// Mitsubishi GX Works2 project: PLC_Group7 Finishhh   PLC: FX3G

// global labels: Global1
VAR_GLOBAL
  Start_Day AT X007 : BOOL;
  Emergency_Switch AT X005 : BOOL;
  LackMaterials AT M1 : BOOL;
  Work_Day AT Y007 : BOOL;
  Y7coil AT Y007 : BOOL;
  EndDayReset AT M2 : BOOL;
  Chocolate_Input AT D1100 : REAL;
  Chocolate_Stock AT D1101 : REAL;
  Nuts_Input AT D1102 : REAL;
  Nuts_Stock AT D1103 : REAL;
  Fistock_Input AT D1104 : REAL;
  Fistock_Stock AT D1105 : REAL;
  Kadaif_Input AT D1106 : REAL;
  Kadaif_Stock AT D1107 : REAL;
  Chocolate_Package AT D1108 : REAL;
  Start_Melting AT X001 : BOOL;
  Min_Chocolate AT E400 : REAL;
  Check_Chocolate AT M3 : BOOL;
  Chocolate_Melting_Tank AT D1110 : REAL;
  Temp_Sensor AT X002 : BOOL;
  End_Melting AT Y001 : BOOL;
  Flag_End_Melting AT M4 : BOOL;
  Location_Sensor AT X003 : BOOL;
  Flag_End_Location AT M5 : BOOL;
  MoldCastingTimer AT TC1 : BOOL;
  MoldCasting AT K40 : INT;
  FinishCasting AT TS1 : BOOL;
  InCastingProcess AT Y002 : BOOL;
  Empty_Mold_Tank AT D1114 : REAL;
  Flag_End_Casting AT M6 : BOOL;
  Chocolate_Type AT X004 : BOOL;
  Make_Nuts_Chocolate AT M7 : BOOL;
  Nuts_N AT E100 : REAL;
  Fistock_N AT E100 : REAL;
  Kadaif_N AT E0 : REAL;
  Out_Of_Stock_Nuts AT M9 : BOOL;
  Choose_Type AT X004 : BOOL;
  Dubai_Chocolate AT M8 : BOOL;
  Nuts_D AT E20 : REAL;
  Fistock_D AT E120 : REAL;
  Kadaif_D AT E60 : REAL;
  Out_Of_Stock_Dubai AT M10 : BOOL;
  Start_Making AT X004 : BOOL;
END_VAR
VAR_GLOBAL CONSTANT
  Convert : REAL := 400;
END_VAR
VAR_GLOBAL
  Chocolate_Ch AT D7000 : REAL;
  Chocolate_Choice AT D7000 : REAL;
  Choose_Nuts AT E5 : REAL;
  Make_Dubai_Chocolate AT M8 : BOOL;
  Min_Amount_Nuts_D AT E10 : REAL;
  Amount_Cream_Nuts AT E50 : REAL;
  Cream_Tank_Nuts AT D1116 : REAL;
  Cream_Tank_Dubi AT D1118 : REAL;
  Amount_Cream_Dubai AT E50 : REAL;
  Cream_Tank_Dubai AT D1118 : REAL;
  Start_Cream AT M11 : BOOL;
  Start_Flash AT TC2 : BOOL;
  Finish_Flesh AT TS2 : BOOL;
  Start_Flashing AT M12 : BOOL;
  Timer_Flash AT K50 : INT;
  Flech3 AT TC3 : BOOL;
  Flesh_CreaFill3 AT Y003 : BOOL;
  Finish_Flesh3 AT TS3 : BOOL;
  Flesh4 AT TC4 : BOOL;
  Finish_Flesh4 AT TS4 : BOOL;
  Flesh_CreamFill4 AT Y004 : BOOL;
  Flesh_CreamFill3 AT Y003 : BOOL;
  Time_Flesh34 AT K5 : INT;
  Melting AT Y001 : BOOL;
  Freeze_Chocolate AT X006 : BOOL;
  Time_Freeze AT TC5 : BOOL;
  Three_Sec_Freeze AT K30 : INT;
  Freeze_Light AT Y006 : BOOL;
  Finish_Freeze AT TS5 : BOOL;
  Start_Packing AT X006 : BOOL;
  Chocolate_Counter AT CC1 : BOOL;
  Chocolate_Package_Counter AT CC1 : BOOL;
END_VAR
VAR_GLOBAL CONSTANT
  Four_Package_Chocolate : INT := K4;
END_VAR
VAR_GLOBAL
  Packing_One AT X000 : BOOL;
  Pack_Light AT Y005 : BOOL;
  CS_Packing AT CS1 : BOOL;
  Counter_1 AT K1 : INT;
  Package_Number AT D4000 : REAL;
  Package_Number_Output : INT;
END_VAR
VAR_GLOBAL CONSTANT
  PI : INT := 40;
END_VAR
VAR_GLOBAL
  Analog_Output AT D8282 : INT;
  Insert_Stock AT M14 : BOOL;
  Analog_Input AT D8280 : INT;
  Analog_Input1 AT D8280 : INT;
  Choose_Nuts1 AT E5 : REAL;
  Amount_Cream_Dubai1 AT E200 : REAL;
  Amount_Cream_Nuts1 AT E200 : REAL;
  Flash_Help AT M15 : BOOL;
END_VAR
VAR_GLOBAL CONSTANT
  PI1 : INT := 40;
END_VAR
VAR_GLOBAL
  Out_Of_Stock AT M9 : BOOL;
END_VAR
VAR_GLOBAL CONSTANT
  Zero : REAL;
END_VAR
VAR_GLOBAL
  Reset_Data AT X010 : BOOL;
END_VAR

// task Task_01 (event TRUE, interval 0, priority 31): POU_01

PROGRAM POU_01
(* structured ladder/FBD written out as ST: instructions are called as NAME(EN, inputs, outputs); _pN, _eN, _tN stand for wires *)
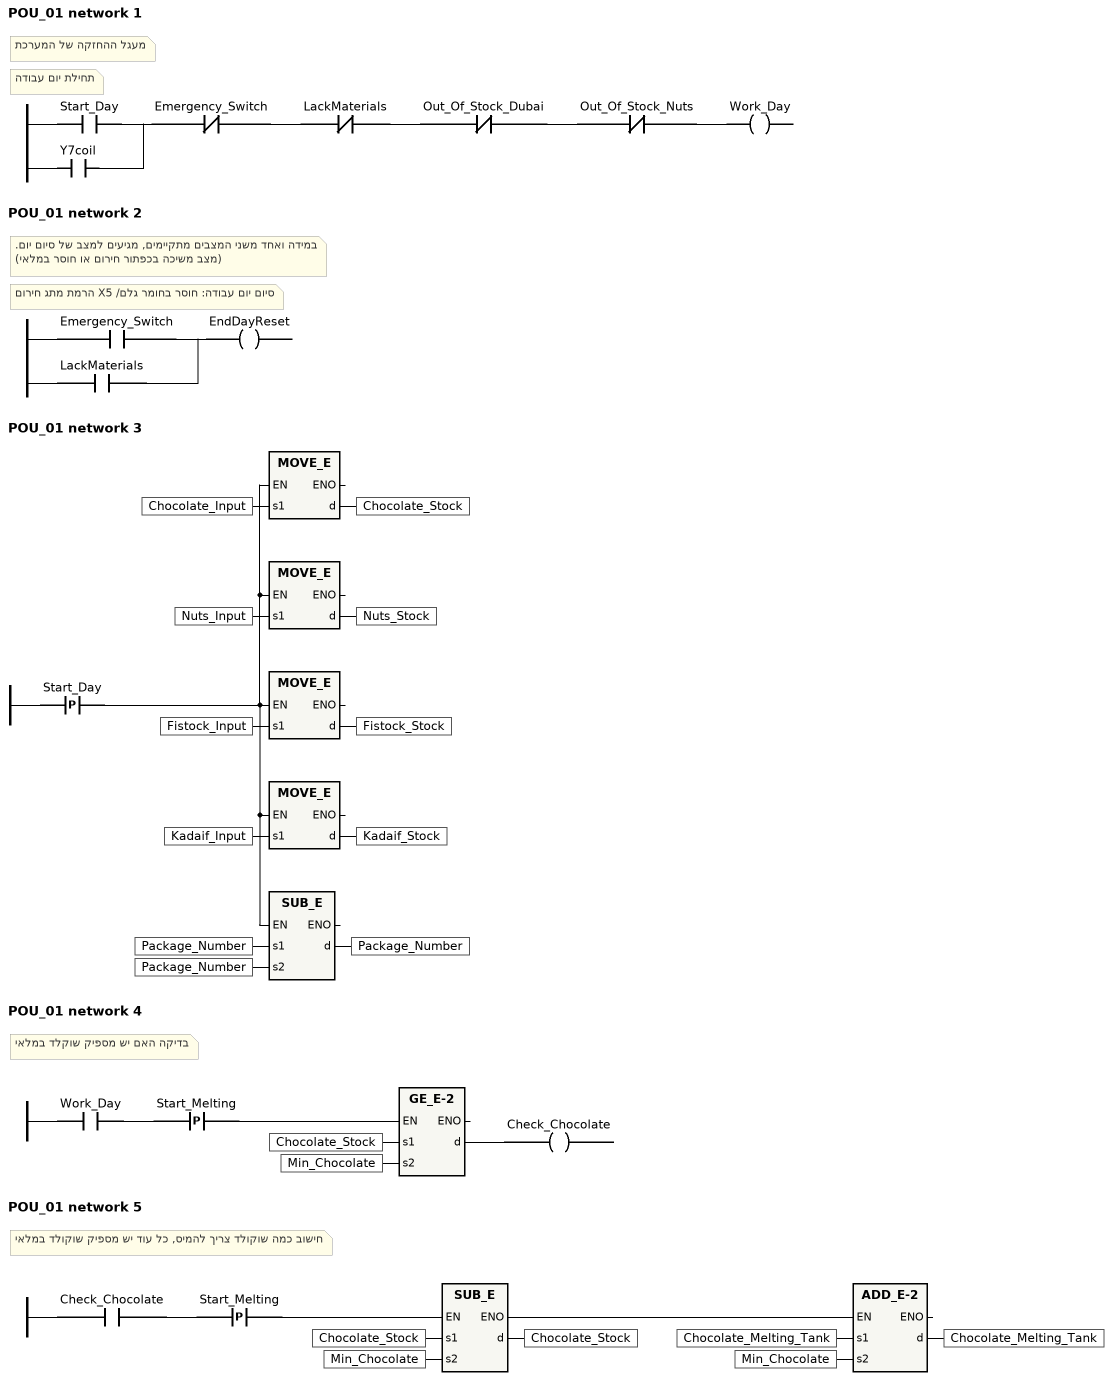
(* network 1 מעגל ההחזקה של המערכ *)
(* מעגל ההחזקה של המערכת *)
(* תחילת יום עבודה *)
Work_Day := ((((Start_Day OR Y7coil) AND NOT Emergency_Switch) AND NOT LackMaterials) AND NOT Out_Of_Stock_Dubai) AND NOT Out_Of_Stock_Nuts;
(* network 2 *)
(* במידה ואחד משני המצבים מתקיימים, מגיעים למצב של סיום יום. (מצב משיכה בכפתור חירום או חוסר במלאי) *)
(* סיום יום עבודה: חוסר בחומר גלם/ X5 הרמת מתג חירום *)
EndDayReset := Emergency_Switch OR LackMaterials;
(* network 3 *)
_p1 := LDP(TRUE, Start_Day);
MOVE_E(_p1, Chocolate_Input, Chocolate_Stock);
MOVE_E(_p1, Nuts_Input, Nuts_Stock);
MOVE_E(_p1, Fistock_Input, Fistock_Stock);
MOVE_E(_p1, Kadaif_Input, Kadaif_Stock);
SUB_E(_p1, Package_Number, Package_Number, Package_Number);
(* network 4 *)
(* בדיקה האם יש מספיק שוקלד במלאי *)
GE_E(Work_Day AND LDP(TRUE, Start_Melting), Chocolate_Stock, Min_Chocolate, _t1);
Check_Chocolate := _t1;
(* network 5 *)
(* חישוב כמה שוקולד צריך להמיס, כל עוד יש מספיק שוקולד במלאי *)
_e1 := SUB_E(Check_Chocolate AND LDP(TRUE, Start_Melting), Chocolate_Stock, Min_Chocolate, Chocolate_Stock);
ADD_E(_e1, Chocolate_Melting_Tank, Min_Chocolate, Chocolate_Melting_Tank);
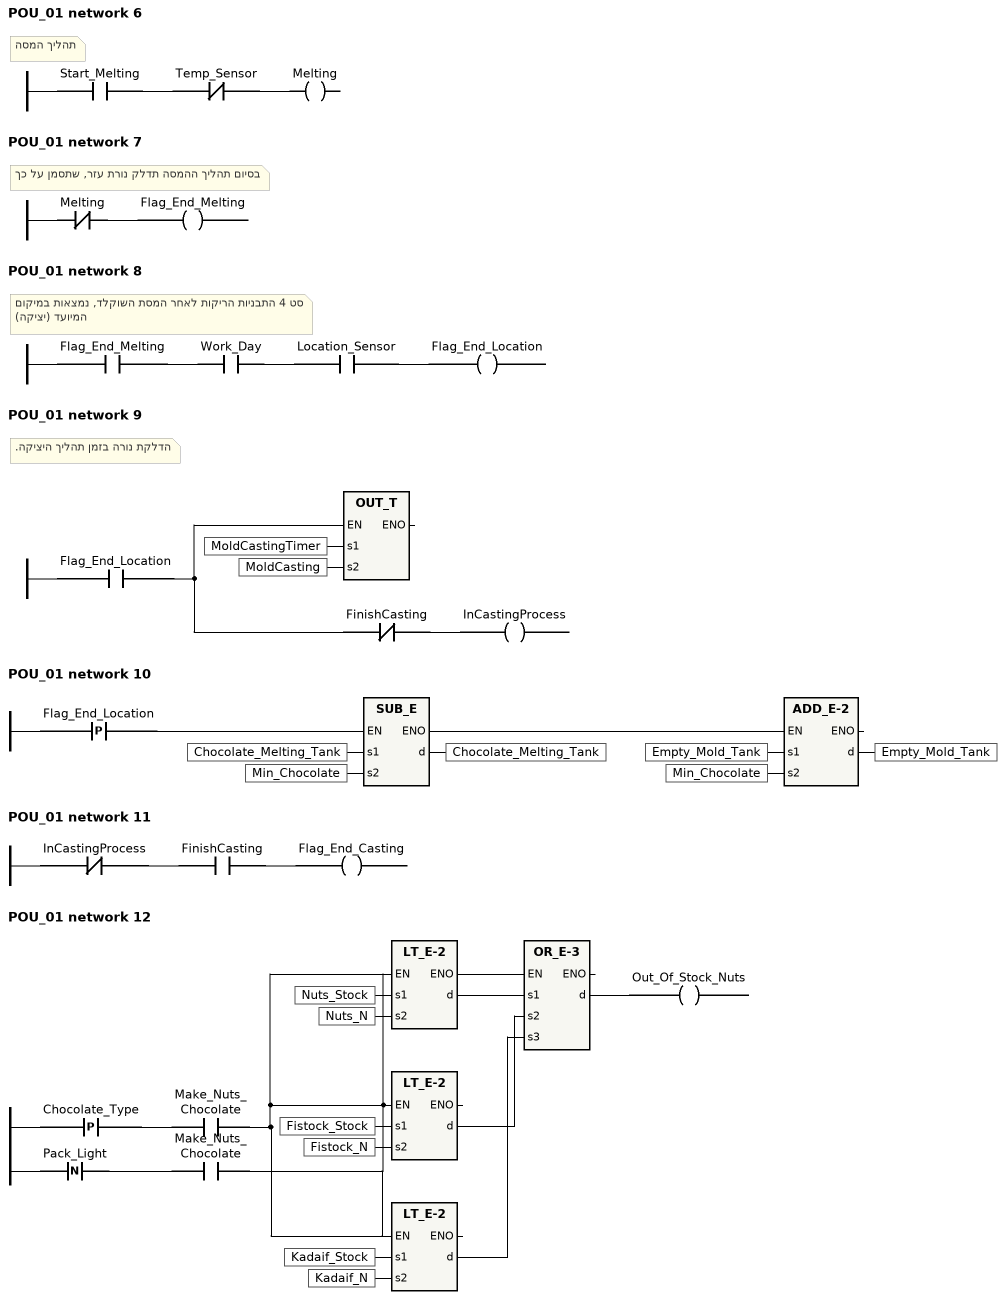
(* network 6 *)
(* תהליך המסה *)
Melting := Start_Melting AND NOT Temp_Sensor;
(* network 7 *)
(* בסיום תהליך ההמסה תדלק נורת עזר, שתסמן על כך *)
Flag_End_Melting := NOT Melting;
(* network 8 *)
(* סט 4 התבניות הריקות לאחר המסת השוקלד, נמצאות במיקום המיועד (יציקה) *)
Flag_End_Location := Flag_End_Melting AND Work_Day AND Location_Sensor;
(* network 9 *)
(* הדלקת נורה בזמן תהליך היציקה. *)
OUT_T(Flag_End_Location, MoldCastingTimer, MoldCasting);
InCastingProcess := Flag_End_Location AND NOT FinishCasting;
(* network 10 *)
_e1 := SUB_E(LDP(TRUE, Flag_End_Location), Chocolate_Melting_Tank, Min_Chocolate, Chocolate_Melting_Tank);
ADD_E(_e1, Empty_Mold_Tank, Min_Chocolate, Empty_Mold_Tank);
(* network 11 *)
Flag_End_Casting := NOT InCastingProcess AND FinishCasting;
(* network 12 *)
_p1 := (LDP(TRUE, Chocolate_Type) AND Make_Nuts_Chocolate) OR (LDF(TRUE, Pack_Light) AND Make_Nuts_Chocolate);
_e3 := LT_E(_p1, Nuts_Stock, Nuts_N, _t2);
LT_E(_p1, Fistock_Stock, Fistock_N, _t4);
LT_E(_p1, Kadaif_Stock, Kadaif_N, _t5);
OR_E(_e3, _t2, _t4, _t5, _t6);
Out_Of_Stock_Nuts := _t6;
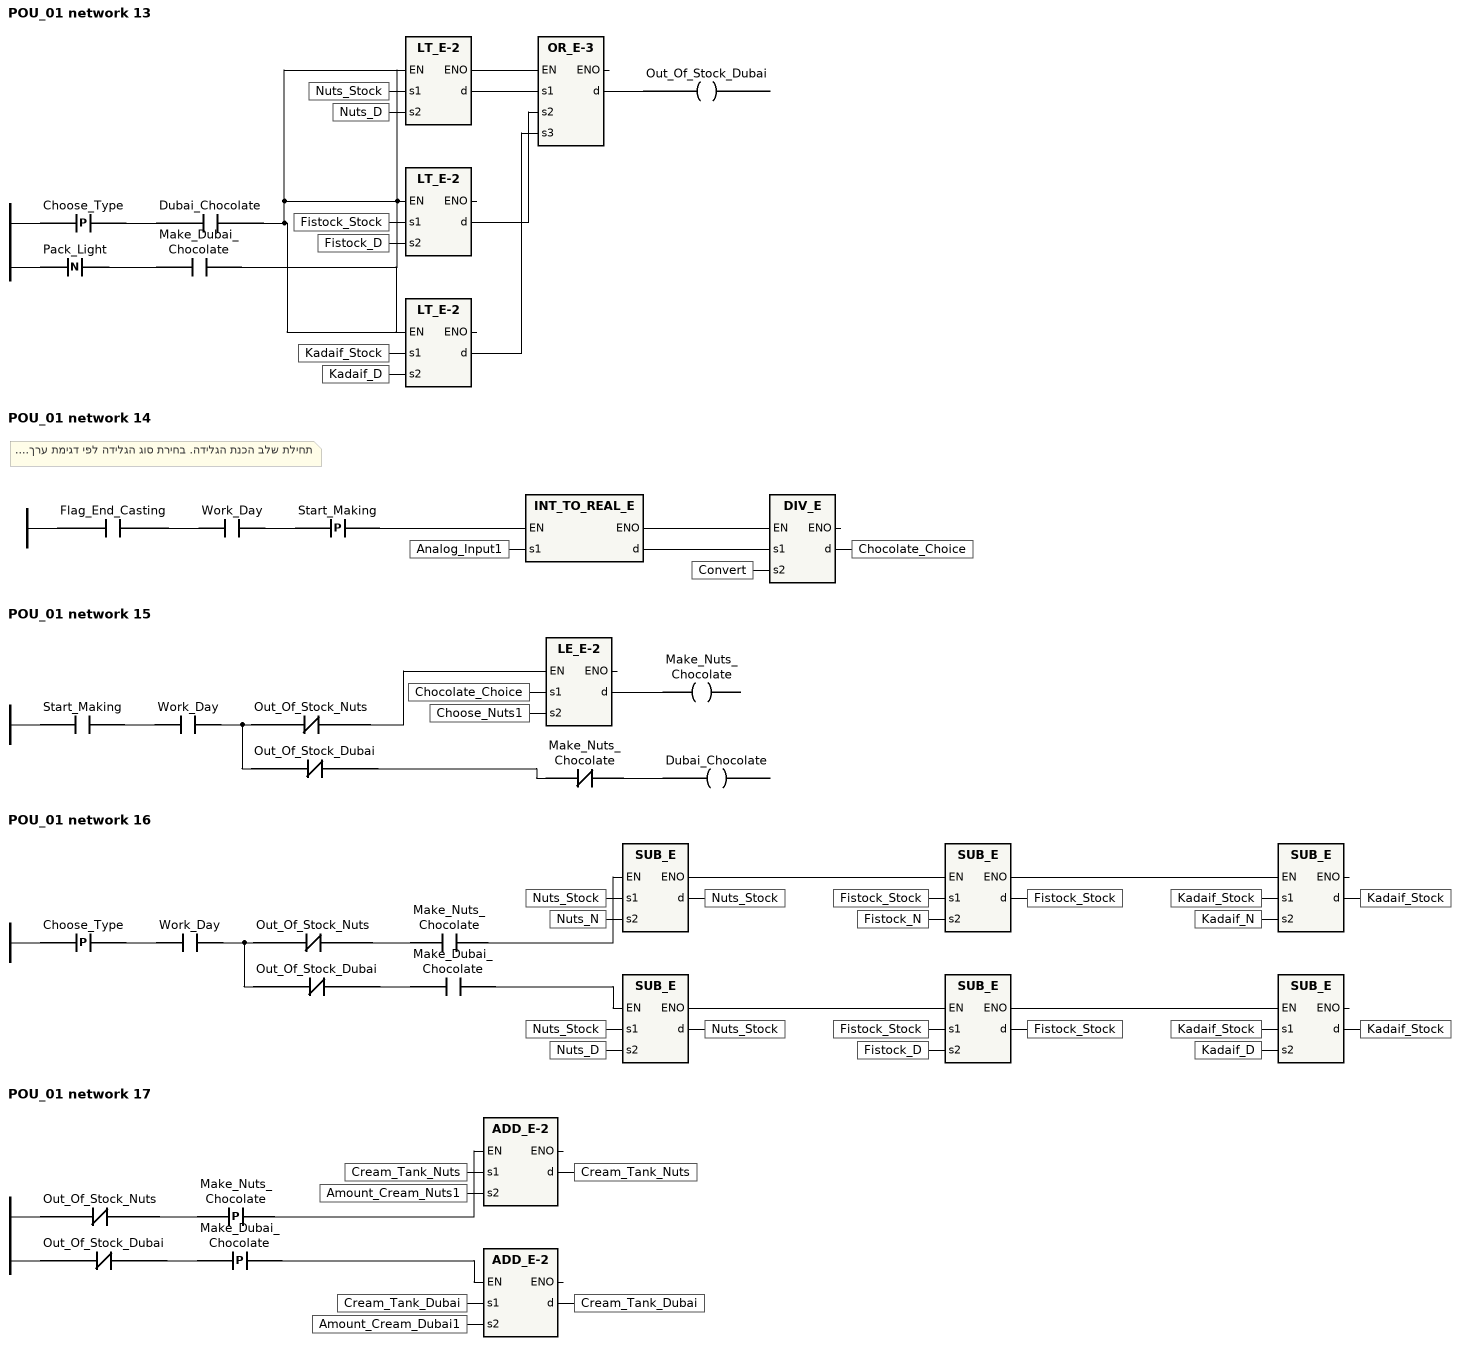
(* network 13 *)
_p1 := (LDP(TRUE, Choose_Type) AND Dubai_Chocolate) OR (LDF(TRUE, Pack_Light) AND Make_Dubai_Chocolate);
_e3 := LT_E(_p1, Nuts_Stock, Nuts_D, _t2);
LT_E(_p1, Fistock_Stock, Fistock_D, _t4);
LT_E(_p1, Kadaif_Stock, Kadaif_D, _t5);
OR_E(_e3, _t2, _t4, _t5, _t6);
Out_Of_Stock_Dubai := _t6;
(* network 14 *)
(* תחילת שלב הכנת הגלידה. בחירת סוג הגלידה לפי דגימת ערך.... *)
_e2 := INT_TO_REAL_E(Flag_End_Casting AND Work_Day AND LDP(TRUE, Start_Making), Analog_Input1, _t1);
DIV_E(_e2, _t1, Convert, Chocolate_Choice);
(* network 15 *)
_p1 := Start_Making AND Work_Day;
LE_E(_p1 AND NOT Out_Of_Stock_Nuts, Chocolate_Choice, Choose_Nuts1, _t2);
Make_Nuts_Chocolate := _t2;
Dubai_Chocolate := _p1 AND NOT Out_Of_Stock_Dubai AND NOT Make_Nuts_Chocolate;
(* network 16 *)
_p1 := LDP(TRUE, Choose_Type) AND Work_Day;
_e2 := SUB_E(_p1 AND NOT Out_Of_Stock_Nuts AND Make_Nuts_Chocolate, Nuts_Stock, Nuts_N, Nuts_Stock);
_e3 := SUB_E(_e2, Fistock_Stock, Fistock_N, Fistock_Stock);
SUB_E(_e3, Kadaif_Stock, Kadaif_N, Kadaif_Stock);
_e4 := SUB_E(_p1 AND NOT Out_Of_Stock_Dubai AND Make_Dubai_Chocolate, Nuts_Stock, Nuts_D, Nuts_Stock);
_e5 := SUB_E(_e4, Fistock_Stock, Fistock_D, Fistock_Stock);
SUB_E(_e5, Kadaif_Stock, Kadaif_D, Kadaif_Stock);
(* network 17 *)
ADD_E(NOT Out_Of_Stock_Nuts AND LDP(TRUE, Make_Nuts_Chocolate), Cream_Tank_Nuts, Amount_Cream_Nuts1, Cream_Tank_Nuts);
ADD_E(NOT Out_Of_Stock_Dubai AND LDP(TRUE, Make_Dubai_Chocolate), Cream_Tank_Dubai, Amount_Cream_Dubai1, Cream_Tank_Dubai);
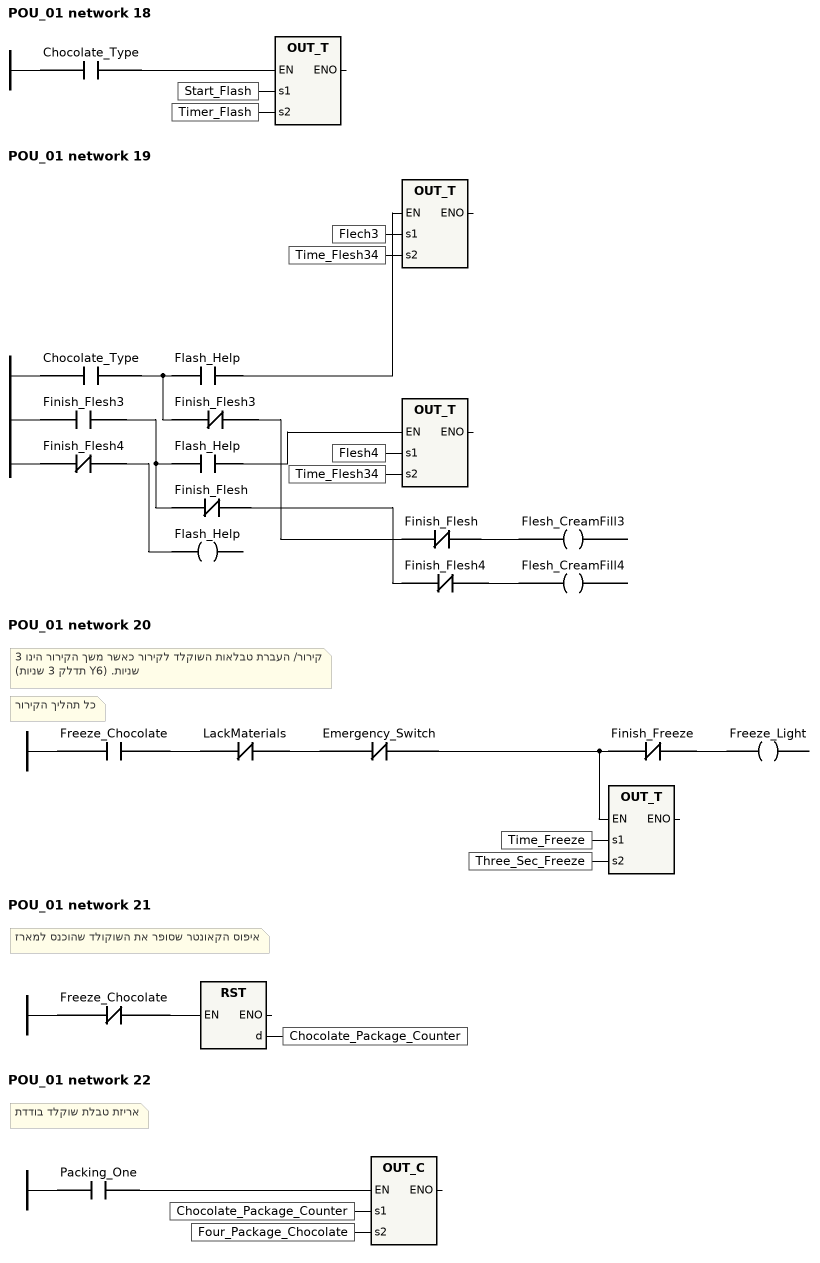
(* network 18 *)
OUT_T(Chocolate_Type, Start_Flash, Timer_Flash);
(* network 19 *)
OUT_T(Chocolate_Type AND Flash_Help, Flech3, Time_Flesh34);
Flesh_CreamFill3 := Chocolate_Type AND NOT Finish_Flesh3 AND NOT Finish_Flesh;
OUT_T(Finish_Flesh3 AND Flash_Help, Flesh4, Time_Flesh34);
Flesh_CreamFill4 := Finish_Flesh3 AND NOT Finish_Flesh AND NOT Finish_Flesh4;
Flash_Help := NOT Finish_Flesh4;
(* network 20 *)
(* קירור/ העברת טבלאות השוקלד לקירור כאשר משך הקירור הינו 3 שניות. (Y6 תדלק 3 שניות) *)
(* כל תהליך הקירור *)
_p1 := Freeze_Chocolate AND NOT LackMaterials AND NOT Emergency_Switch;
Freeze_Light := _p1 AND NOT Finish_Freeze;
OUT_T(_p1, Time_Freeze, Three_Sec_Freeze);
(* network 21 *)
(* איפוס הקאונטר שסופר את השוקולד שהוכנס למארז *)
RST(NOT Freeze_Chocolate, Chocolate_Package_Counter);
(* network 22 *)
(* אריזת טבלת שוקלד בודדת *)
OUT_C(Packing_One, Chocolate_Package_Counter, Four_Package_Chocolate);
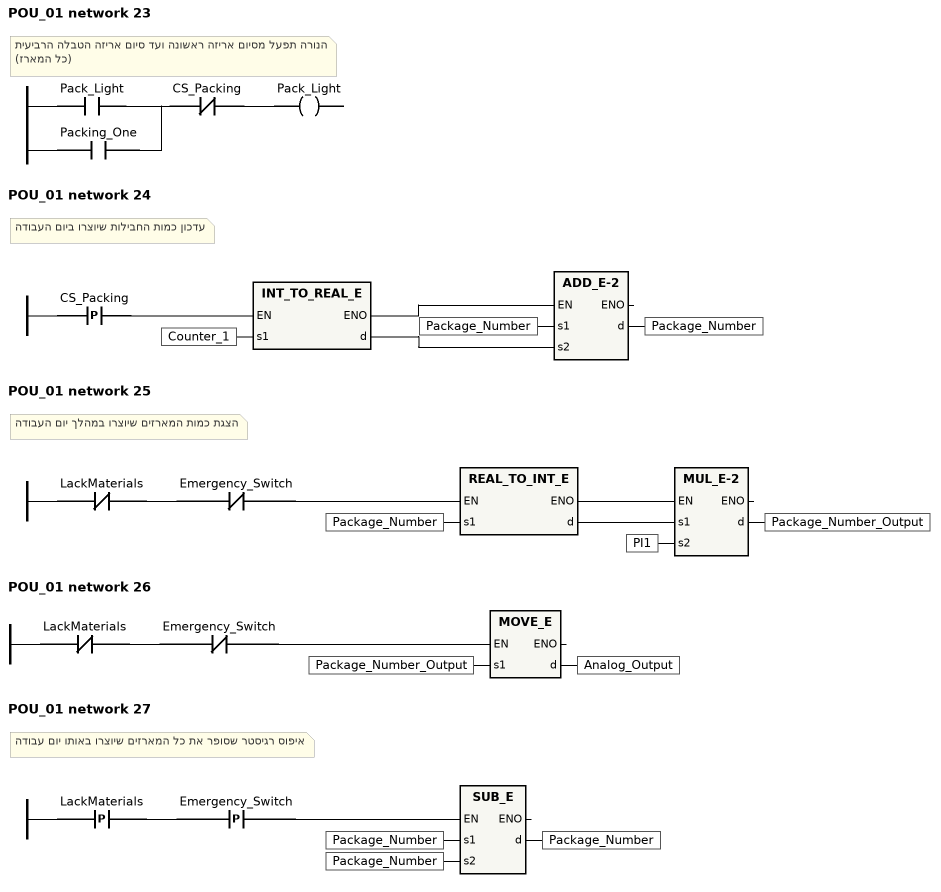
(* network 23 *)
(* הנורה תפעל מסיום אריזה ראשונה ועד סיום אריזה הטבלה הרביעית (כל המארז) *)
Pack_Light := (Pack_Light OR Packing_One) AND NOT CS_Packing;
(* network 24 *)
(* עדכון כמות החבילות שיוצרו ביום העבודה *)
_e2 := INT_TO_REAL_E(LDP(TRUE, CS_Packing), Counter_1, _t1);
ADD_E(_e2, Package_Number, _t1, Package_Number);
(* network 25 *)
(* הצגת כמות המארזים שיוצרו במהלך יום העבודה *)
_e2 := REAL_TO_INT_E(NOT LackMaterials AND NOT Emergency_Switch, Package_Number, _t1);
MUL_E(_e2, _t1, PI1, Package_Number_Output);
(* network 26 *)
MOVE_E(NOT LackMaterials AND NOT Emergency_Switch, Package_Number_Output, Analog_Output);
(* network 27 *)
(* איפוס רגיסטר שסופר את כל המארזים שיוצרו באותו יום עבודה *)
SUB_E(LDP(TRUE, LackMaterials) AND LDP(TRUE, Emergency_Switch), Package_Number, Package_Number, Package_Number);
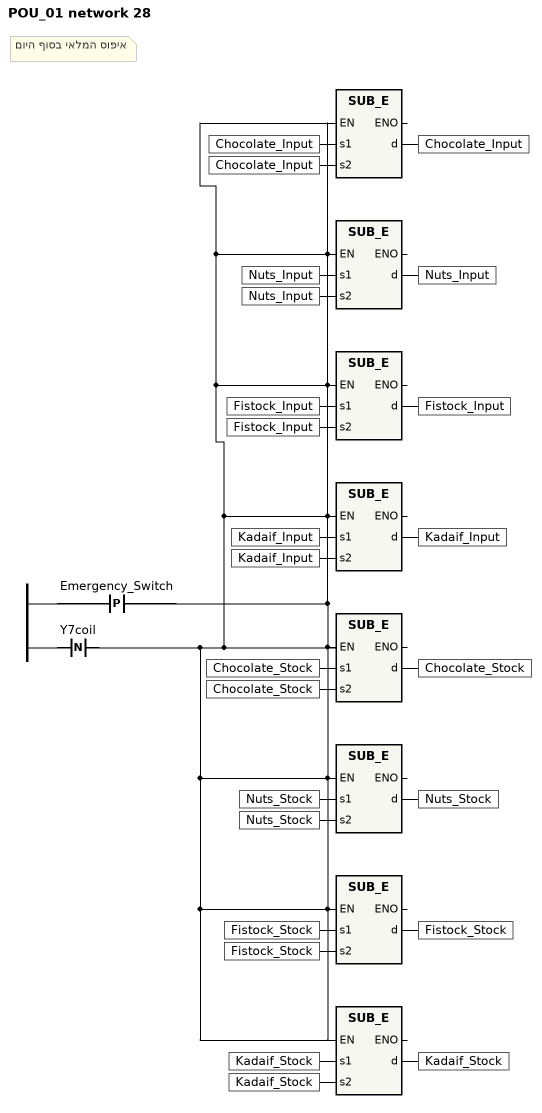
(* network 28 *)
(* איפוס המלאי בסוף היום *)
_p1 := LDP(TRUE, Emergency_Switch) OR LDF(TRUE, Y7coil);
SUB_E(_p1, Chocolate_Input, Chocolate_Input, Chocolate_Input);
SUB_E(_p1, Nuts_Input, Nuts_Input, Nuts_Input);
SUB_E(_p1, Fistock_Input, Fistock_Input, Fistock_Input);
SUB_E(_p1, Kadaif_Input, Kadaif_Input, Kadaif_Input);
SUB_E(_p1, Chocolate_Stock, Chocolate_Stock, Chocolate_Stock);
SUB_E(_p1, Nuts_Stock, Nuts_Stock, Nuts_Stock);
SUB_E(_p1, Fistock_Stock, Fistock_Stock, Fistock_Stock);
SUB_E(_p1, Kadaif_Stock, Kadaif_Stock, Kadaif_Stock);
END_PROGRAM
